(* Logix 5000 project; controller RN21_Architecture 1769-L16ER-BB1B rev 35.11; software revision 35.00; part 5 of 9 *)
(* tags used below, declared in another part *)
   AUDSrc : UDT_Audit;
   RN21_AUD_BAMTrig : DINT[5];
   RN21_AUD_BAT_NTrig : DINT[4];
   RN21_AUD_BAT_PTrig : DINT[4];
   RN21_AUD_NEG_ONS : BOOL[128];
   RN21_AUD_POS_ONS : BOOL[128];
   RN21_AUDBAM_ONS : BOOL[128];
   RN21_Map_BAM : BOOL[128];
   RN21_Map_BAT : BOOL[32];
   RN21_MapBAT_OB : BOOL[128];
(* MainProgram, continued *)

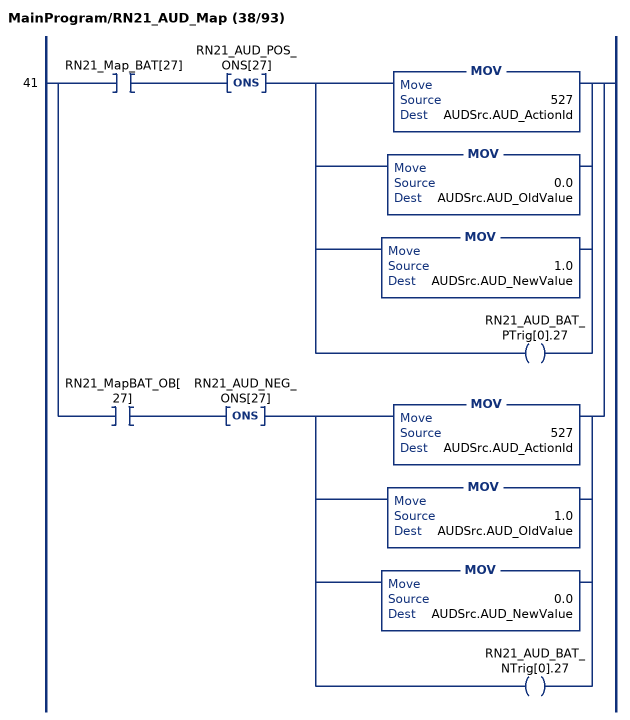
   [picture p120: MainProgram/RN21_AUD_Map rungs 41-41]
   41: [XIC(RN21_Map_BAT[27]) ONS(RN21_AUD_POS_ONS[27]) [MOV(527,AUDSrc.AUD_ActionId) ,MOV(0.0,AUDSrc.AUD_OldValue) ,MOV(1.0,AUDSrc.AUD_NewValue) ,OTE(RN21_AUD_BAT_PTrig[0].27) ] ,XIC(RN21_MapBAT_OB[27]) ONS(RN21_AUD_NEG_ONS[27]) [MOV(527,AUDSrc.AUD_ActionId) ,MOV(1.0,AUDSrc.AUD_OldValue) ,MOV(0.0,AUDSrc.AUD_NewValue) ,OTE(RN21_AUD_BAT_NTrig[0].27) ] ];
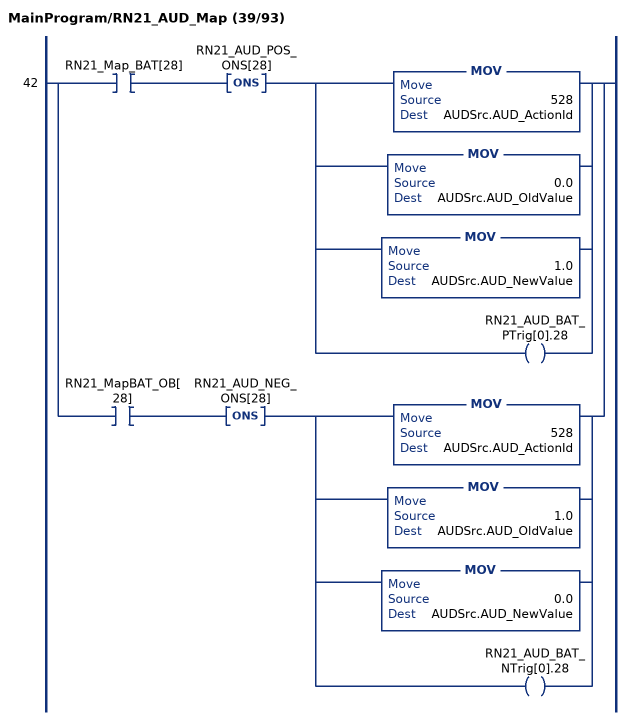
   42: [XIC(RN21_Map_BAT[28]) ONS(RN21_AUD_POS_ONS[28]) [MOV(528,AUDSrc.AUD_ActionId) ,MOV(0.0,AUDSrc.AUD_OldValue) ,MOV(1.0,AUDSrc.AUD_NewValue) ,OTE(RN21_AUD_BAT_PTrig[0].28) ] ,XIC(RN21_MapBAT_OB[28]) ONS(RN21_AUD_NEG_ONS[28]) [MOV(528,AUDSrc.AUD_ActionId) ,MOV(1.0,AUDSrc.AUD_OldValue) ,MOV(0.0,AUDSrc.AUD_NewValue) ,OTE(RN21_AUD_BAT_NTrig[0].28) ] ];
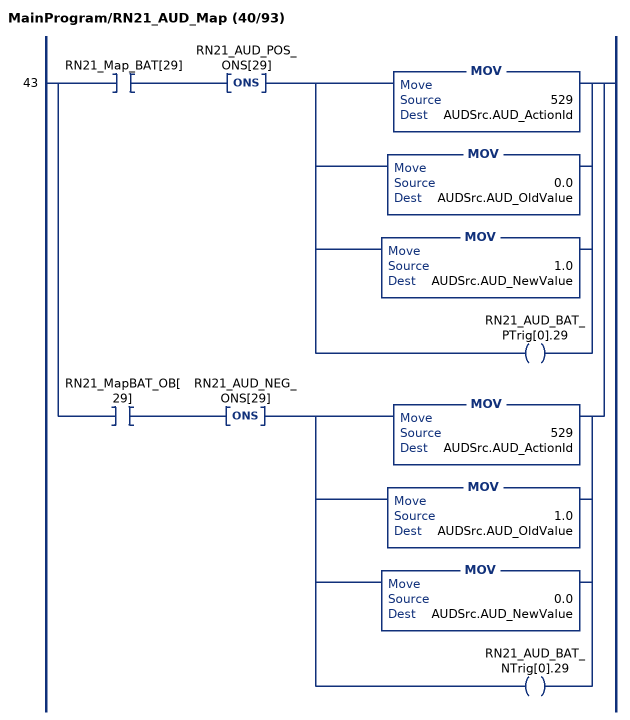
   43: [XIC(RN21_Map_BAT[29]) ONS(RN21_AUD_POS_ONS[29]) [MOV(529,AUDSrc.AUD_ActionId) ,MOV(0.0,AUDSrc.AUD_OldValue) ,MOV(1.0,AUDSrc.AUD_NewValue) ,OTE(RN21_AUD_BAT_PTrig[0].29) ] ,XIC(RN21_MapBAT_OB[29]) ONS(RN21_AUD_NEG_ONS[29]) [MOV(529,AUDSrc.AUD_ActionId) ,MOV(1.0,AUDSrc.AUD_OldValue) ,MOV(0.0,AUDSrc.AUD_NewValue) ,OTE(RN21_AUD_BAT_NTrig[0].29) ] ];
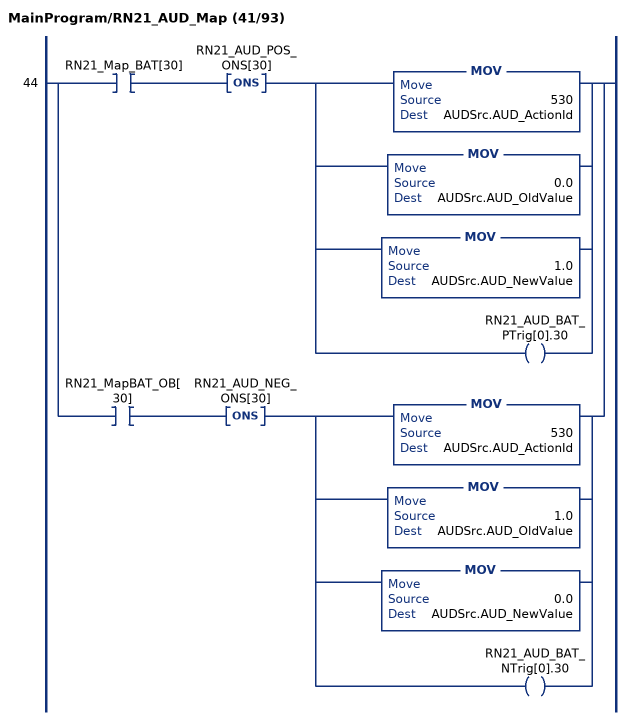
   44: [XIC(RN21_Map_BAT[30]) ONS(RN21_AUD_POS_ONS[30]) [MOV(530,AUDSrc.AUD_ActionId) ,MOV(0.0,AUDSrc.AUD_OldValue) ,MOV(1.0,AUDSrc.AUD_NewValue) ,OTE(RN21_AUD_BAT_PTrig[0].30) ] ,XIC(RN21_MapBAT_OB[30]) ONS(RN21_AUD_NEG_ONS[30]) [MOV(530,AUDSrc.AUD_ActionId) ,MOV(1.0,AUDSrc.AUD_OldValue) ,MOV(0.0,AUDSrc.AUD_NewValue) ,OTE(RN21_AUD_BAT_NTrig[0].30) ] ];
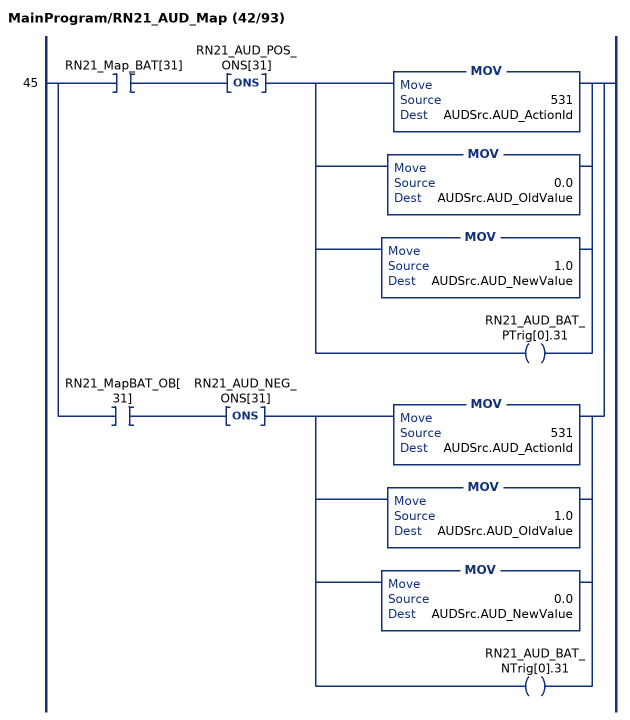
   45: [XIC(RN21_Map_BAT[31]) ONS(RN21_AUD_POS_ONS[31]) [MOV(531,AUDSrc.AUD_ActionId) ,MOV(0.0,AUDSrc.AUD_OldValue) ,MOV(1.0,AUDSrc.AUD_NewValue) ,OTE(RN21_AUD_BAT_PTrig[0].31) ] ,XIC(RN21_MapBAT_OB[31]) ONS(RN21_AUD_NEG_ONS[31]) [MOV(531,AUDSrc.AUD_ActionId) ,MOV(1.0,AUDSrc.AUD_OldValue) ,MOV(0.0,AUDSrc.AUD_NewValue) ,OTE(RN21_AUD_BAT_NTrig[0].31) ] ];
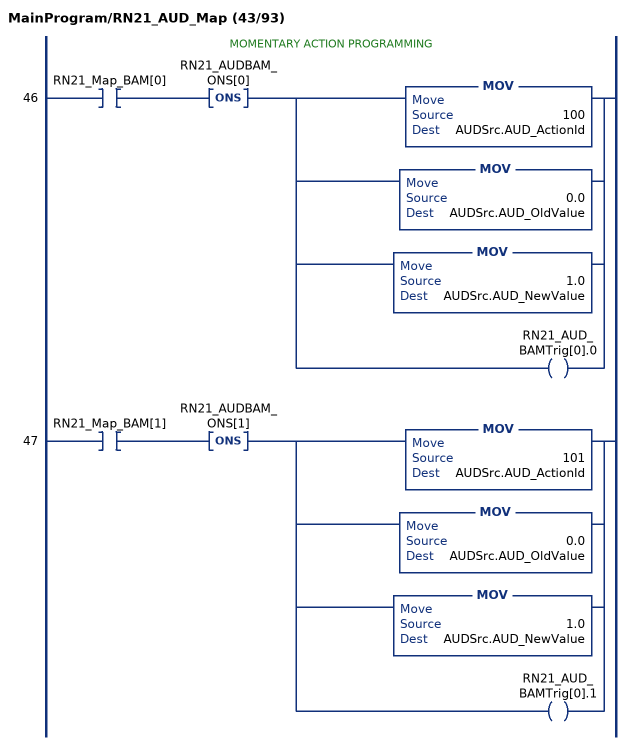
   // MOMENTARY ACTION PROGRAMMING
   46: XIC(RN21_Map_BAM[0])ONS(RN21_AUDBAM_ONS[0])[MOV(100,AUDSrc.AUD_ActionId) ,MOV(0.0,AUDSrc.AUD_OldValue) ,MOV(1.0,AUDSrc.AUD_NewValue) ,OTE(RN21_AUD_BAMTrig[0].0) ];
   47: XIC(RN21_Map_BAM[1])ONS(RN21_AUDBAM_ONS[1])[MOV(101,AUDSrc.AUD_ActionId) ,MOV(0.0,AUDSrc.AUD_OldValue) ,MOV(1.0,AUDSrc.AUD_NewValue) ,OTE(RN21_AUD_BAMTrig[0].1) ];
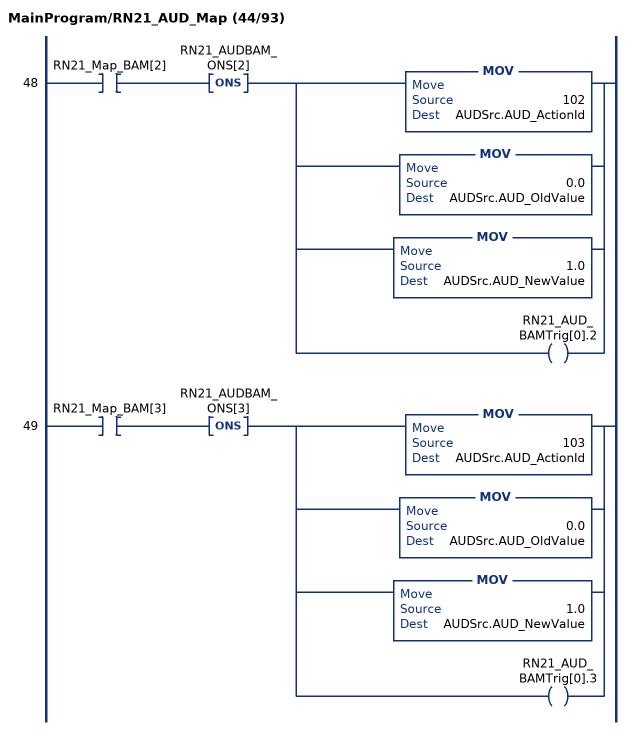
   48: XIC(RN21_Map_BAM[2])ONS(RN21_AUDBAM_ONS[2])[MOV(102,AUDSrc.AUD_ActionId) ,MOV(0.0,AUDSrc.AUD_OldValue) ,MOV(1.0,AUDSrc.AUD_NewValue) ,OTE(RN21_AUD_BAMTrig[0].2) ];
   49: XIC(RN21_Map_BAM[3])ONS(RN21_AUDBAM_ONS[3])[MOV(103,AUDSrc.AUD_ActionId) ,MOV(0.0,AUDSrc.AUD_OldValue) ,MOV(1.0,AUDSrc.AUD_NewValue) ,OTE(RN21_AUD_BAMTrig[0].3) ];
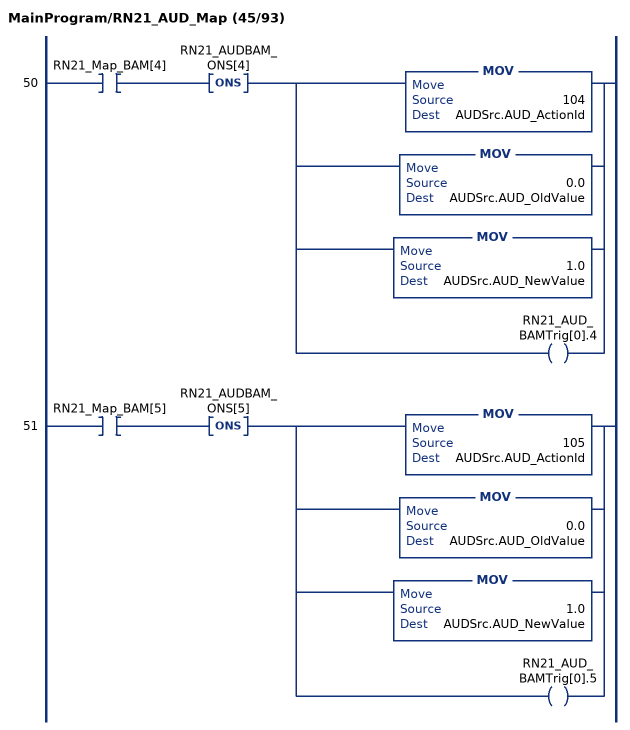
   50: XIC(RN21_Map_BAM[4])ONS(RN21_AUDBAM_ONS[4])[MOV(104,AUDSrc.AUD_ActionId) ,MOV(0.0,AUDSrc.AUD_OldValue) ,MOV(1.0,AUDSrc.AUD_NewValue) ,OTE(RN21_AUD_BAMTrig[0].4) ];
   51: XIC(RN21_Map_BAM[5])ONS(RN21_AUDBAM_ONS[5])[MOV(105,AUDSrc.AUD_ActionId) ,MOV(0.0,AUDSrc.AUD_OldValue) ,MOV(1.0,AUDSrc.AUD_NewValue) ,OTE(RN21_AUD_BAMTrig[0].5) ];
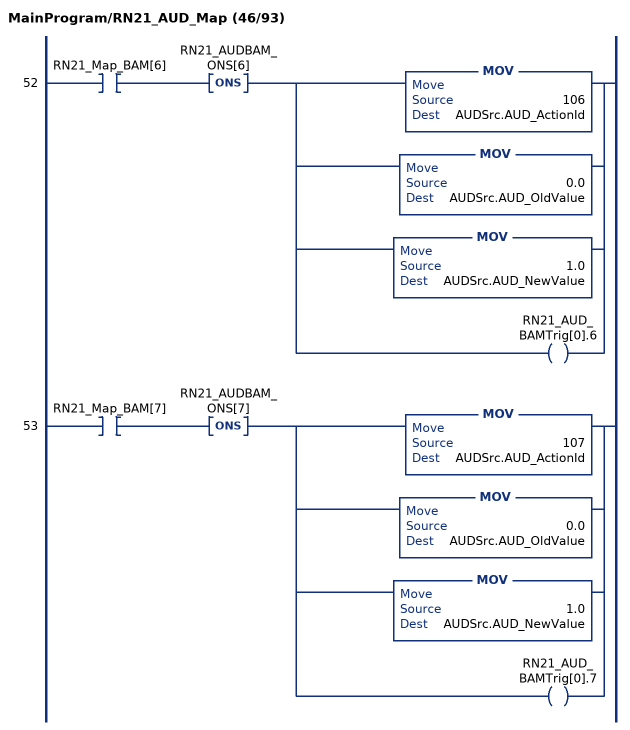
   52: XIC(RN21_Map_BAM[6])ONS(RN21_AUDBAM_ONS[6])[MOV(106,AUDSrc.AUD_ActionId) ,MOV(0.0,AUDSrc.AUD_OldValue) ,MOV(1.0,AUDSrc.AUD_NewValue) ,OTE(RN21_AUD_BAMTrig[0].6) ];
   53: XIC(RN21_Map_BAM[7])ONS(RN21_AUDBAM_ONS[7])[MOV(107,AUDSrc.AUD_ActionId) ,MOV(0.0,AUDSrc.AUD_OldValue) ,MOV(1.0,AUDSrc.AUD_NewValue) ,OTE(RN21_AUD_BAMTrig[0].7) ];
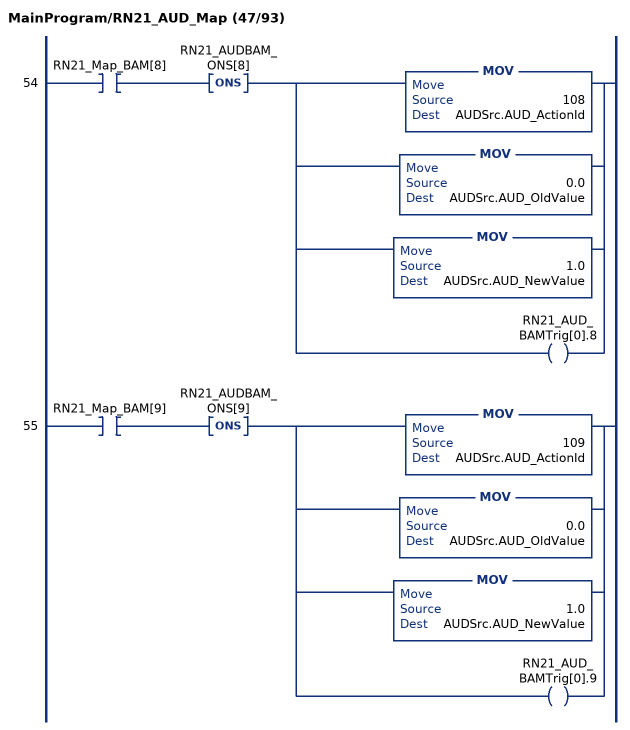
   54: XIC(RN21_Map_BAM[8])ONS(RN21_AUDBAM_ONS[8])[MOV(108,AUDSrc.AUD_ActionId) ,MOV(0.0,AUDSrc.AUD_OldValue) ,MOV(1.0,AUDSrc.AUD_NewValue) ,OTE(RN21_AUD_BAMTrig[0].8) ];
   55: XIC(RN21_Map_BAM[9])ONS(RN21_AUDBAM_ONS[9])[MOV(109,AUDSrc.AUD_ActionId) ,MOV(0.0,AUDSrc.AUD_OldValue) ,MOV(1.0,AUDSrc.AUD_NewValue) ,OTE(RN21_AUD_BAMTrig[0].9) ];
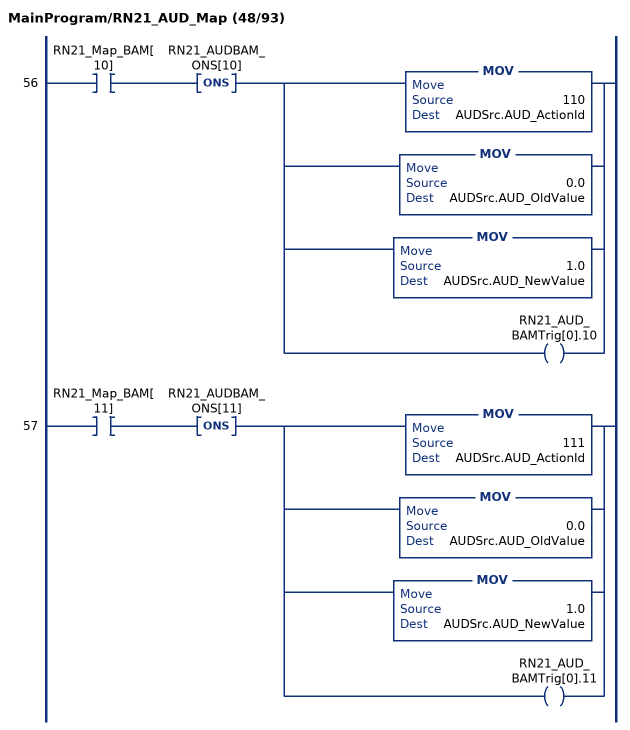
   56: XIC(RN21_Map_BAM[10])ONS(RN21_AUDBAM_ONS[10])[MOV(110,AUDSrc.AUD_ActionId) ,MOV(0.0,AUDSrc.AUD_OldValue) ,MOV(1.0,AUDSrc.AUD_NewValue) ,OTE(RN21_AUD_BAMTrig[0].10) ];
   57: XIC(RN21_Map_BAM[11])ONS(RN21_AUDBAM_ONS[11])[MOV(111,AUDSrc.AUD_ActionId) ,MOV(0.0,AUDSrc.AUD_OldValue) ,MOV(1.0,AUDSrc.AUD_NewValue) ,OTE(RN21_AUD_BAMTrig[0].11) ];
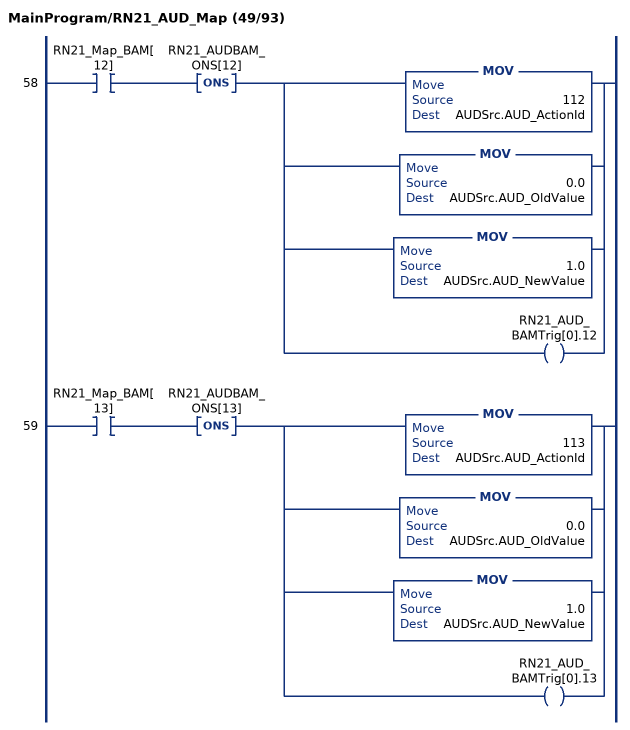
   58: XIC(RN21_Map_BAM[12])ONS(RN21_AUDBAM_ONS[12])[MOV(112,AUDSrc.AUD_ActionId) ,MOV(0.0,AUDSrc.AUD_OldValue) ,MOV(1.0,AUDSrc.AUD_NewValue) ,OTE(RN21_AUD_BAMTrig[0].12) ];
   59: XIC(RN21_Map_BAM[13])ONS(RN21_AUDBAM_ONS[13])[MOV(113,AUDSrc.AUD_ActionId) ,MOV(0.0,AUDSrc.AUD_OldValue) ,MOV(1.0,AUDSrc.AUD_NewValue) ,OTE(RN21_AUD_BAMTrig[0].13) ];
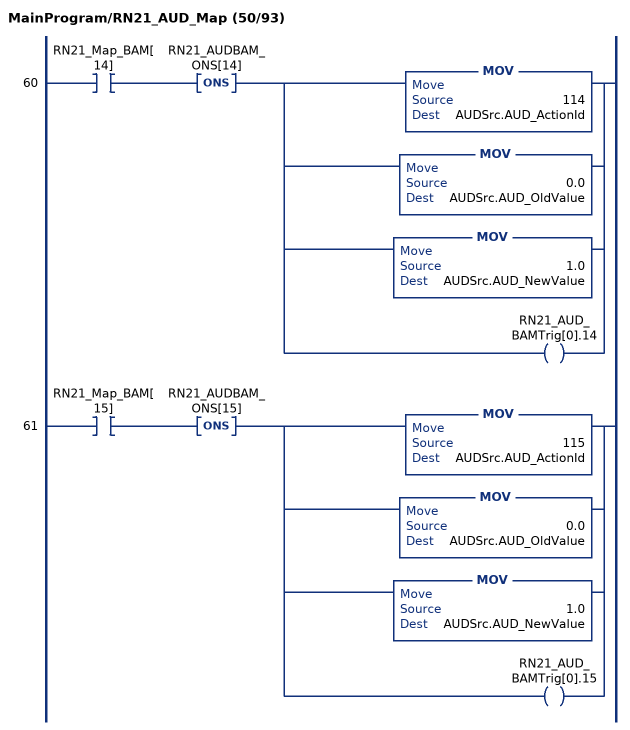
   60: XIC(RN21_Map_BAM[14])ONS(RN21_AUDBAM_ONS[14])[MOV(114,AUDSrc.AUD_ActionId) ,MOV(0.0,AUDSrc.AUD_OldValue) ,MOV(1.0,AUDSrc.AUD_NewValue) ,OTE(RN21_AUD_BAMTrig[0].14) ];
   61: XIC(RN21_Map_BAM[15])ONS(RN21_AUDBAM_ONS[15])[MOV(115,AUDSrc.AUD_ActionId) ,MOV(0.0,AUDSrc.AUD_OldValue) ,MOV(1.0,AUDSrc.AUD_NewValue) ,OTE(RN21_AUD_BAMTrig[0].15) ];
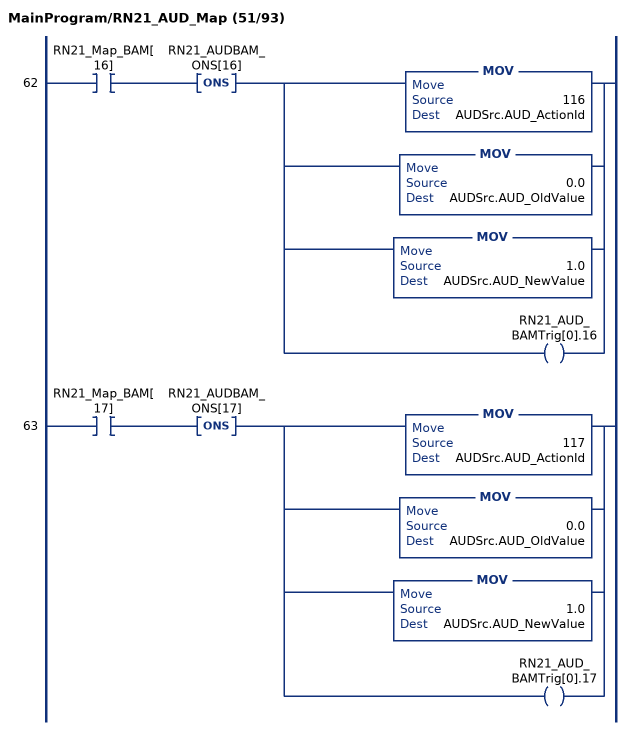
   62: XIC(RN21_Map_BAM[16])ONS(RN21_AUDBAM_ONS[16])[MOV(116,AUDSrc.AUD_ActionId) ,MOV(0.0,AUDSrc.AUD_OldValue) ,MOV(1.0,AUDSrc.AUD_NewValue) ,OTE(RN21_AUD_BAMTrig[0].16) ];
   63: XIC(RN21_Map_BAM[17])ONS(RN21_AUDBAM_ONS[17])[MOV(117,AUDSrc.AUD_ActionId) ,MOV(0.0,AUDSrc.AUD_OldValue) ,MOV(1.0,AUDSrc.AUD_NewValue) ,OTE(RN21_AUD_BAMTrig[0].17) ];
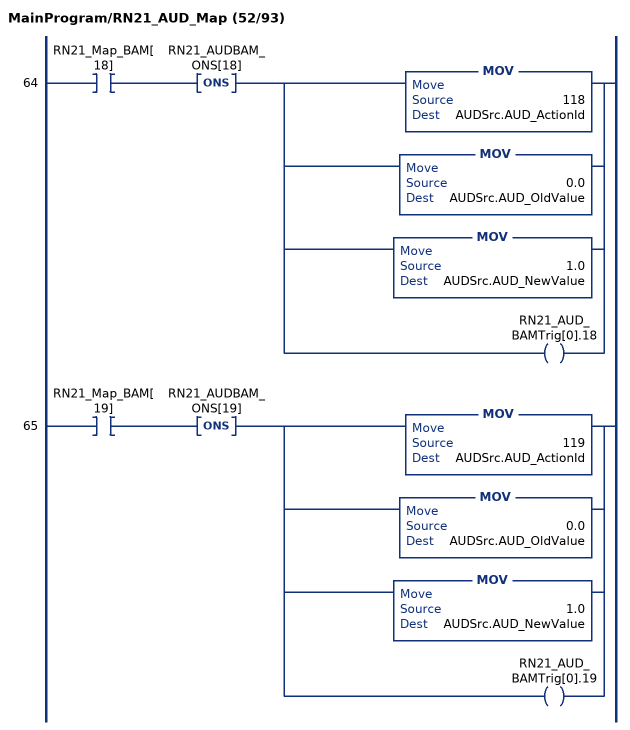
   64: XIC(RN21_Map_BAM[18])ONS(RN21_AUDBAM_ONS[18])[MOV(118,AUDSrc.AUD_ActionId) ,MOV(0.0,AUDSrc.AUD_OldValue) ,MOV(1.0,AUDSrc.AUD_NewValue) ,OTE(RN21_AUD_BAMTrig[0].18) ];
   65: XIC(RN21_Map_BAM[19])ONS(RN21_AUDBAM_ONS[19])[MOV(119,AUDSrc.AUD_ActionId) ,MOV(0.0,AUDSrc.AUD_OldValue) ,MOV(1.0,AUDSrc.AUD_NewValue) ,OTE(RN21_AUD_BAMTrig[0].19) ];
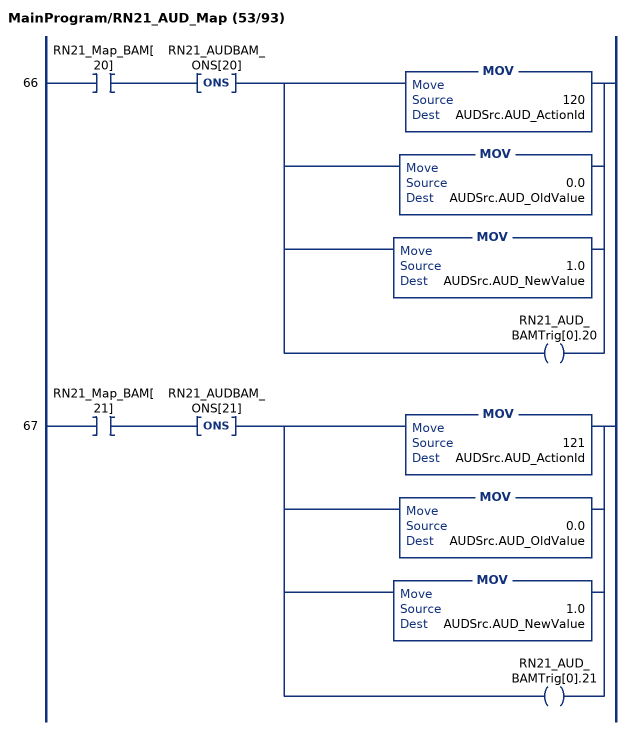
   66: XIC(RN21_Map_BAM[20])ONS(RN21_AUDBAM_ONS[20])[MOV(120,AUDSrc.AUD_ActionId) ,MOV(0.0,AUDSrc.AUD_OldValue) ,MOV(1.0,AUDSrc.AUD_NewValue) ,OTE(RN21_AUD_BAMTrig[0].20) ];
   67: XIC(RN21_Map_BAM[21])ONS(RN21_AUDBAM_ONS[21])[MOV(121,AUDSrc.AUD_ActionId) ,MOV(0.0,AUDSrc.AUD_OldValue) ,MOV(1.0,AUDSrc.AUD_NewValue) ,OTE(RN21_AUD_BAMTrig[0].21) ];
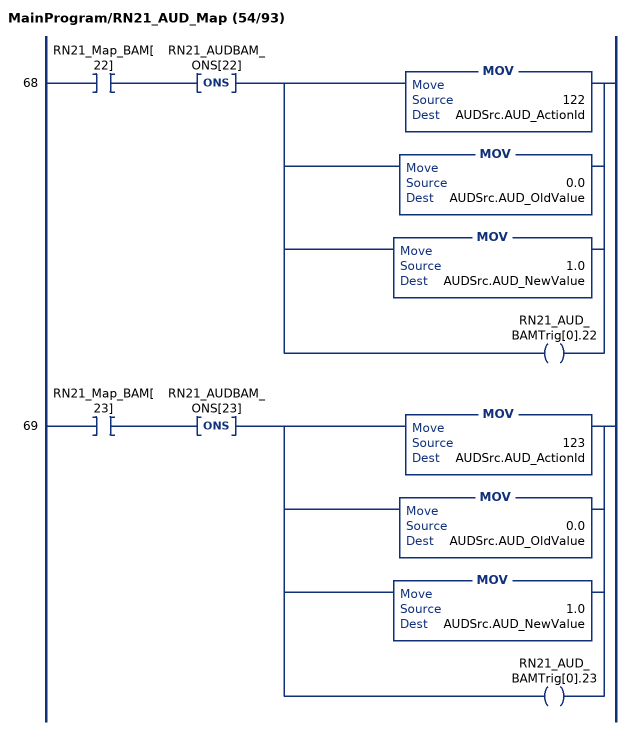
   68: XIC(RN21_Map_BAM[22])ONS(RN21_AUDBAM_ONS[22])[MOV(122,AUDSrc.AUD_ActionId) ,MOV(0.0,AUDSrc.AUD_OldValue) ,MOV(1.0,AUDSrc.AUD_NewValue) ,OTE(RN21_AUD_BAMTrig[0].22) ];
   69: XIC(RN21_Map_BAM[23])ONS(RN21_AUDBAM_ONS[23])[MOV(123,AUDSrc.AUD_ActionId) ,MOV(0.0,AUDSrc.AUD_OldValue) ,MOV(1.0,AUDSrc.AUD_NewValue) ,OTE(RN21_AUD_BAMTrig[0].23) ];
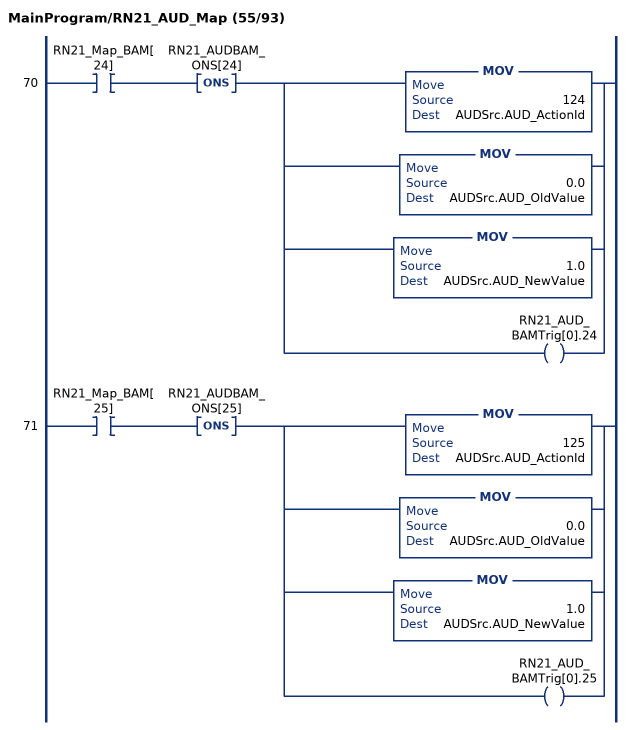
   70: XIC(RN21_Map_BAM[24])ONS(RN21_AUDBAM_ONS[24])[MOV(124,AUDSrc.AUD_ActionId) ,MOV(0.0,AUDSrc.AUD_OldValue) ,MOV(1.0,AUDSrc.AUD_NewValue) ,OTE(RN21_AUD_BAMTrig[0].24) ];
   71: XIC(RN21_Map_BAM[25])ONS(RN21_AUDBAM_ONS[25])[MOV(125,AUDSrc.AUD_ActionId) ,MOV(0.0,AUDSrc.AUD_OldValue) ,MOV(1.0,AUDSrc.AUD_NewValue) ,OTE(RN21_AUD_BAMTrig[0].25) ];
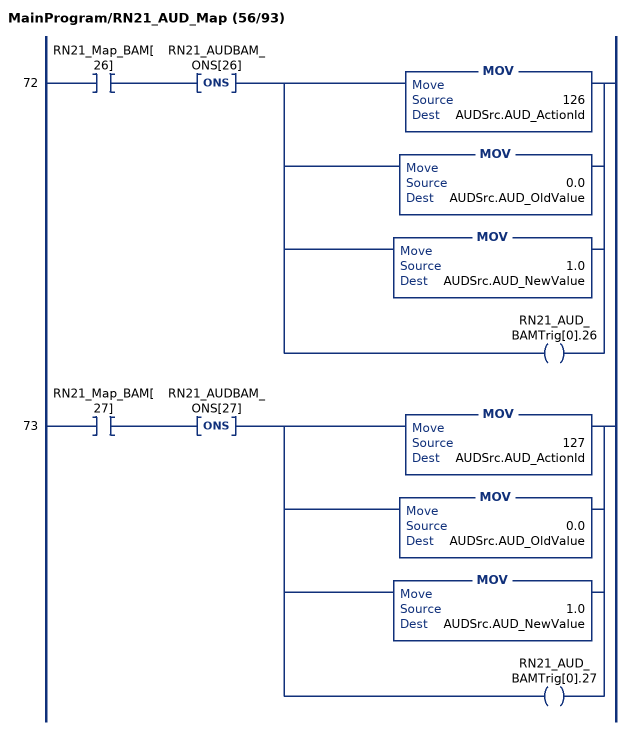
   72: XIC(RN21_Map_BAM[26])ONS(RN21_AUDBAM_ONS[26])[MOV(126,AUDSrc.AUD_ActionId) ,MOV(0.0,AUDSrc.AUD_OldValue) ,MOV(1.0,AUDSrc.AUD_NewValue) ,OTE(RN21_AUD_BAMTrig[0].26) ];
   73: XIC(RN21_Map_BAM[27])ONS(RN21_AUDBAM_ONS[27])[MOV(127,AUDSrc.AUD_ActionId) ,MOV(0.0,AUDSrc.AUD_OldValue) ,MOV(1.0,AUDSrc.AUD_NewValue) ,OTE(RN21_AUD_BAMTrig[0].27) ];
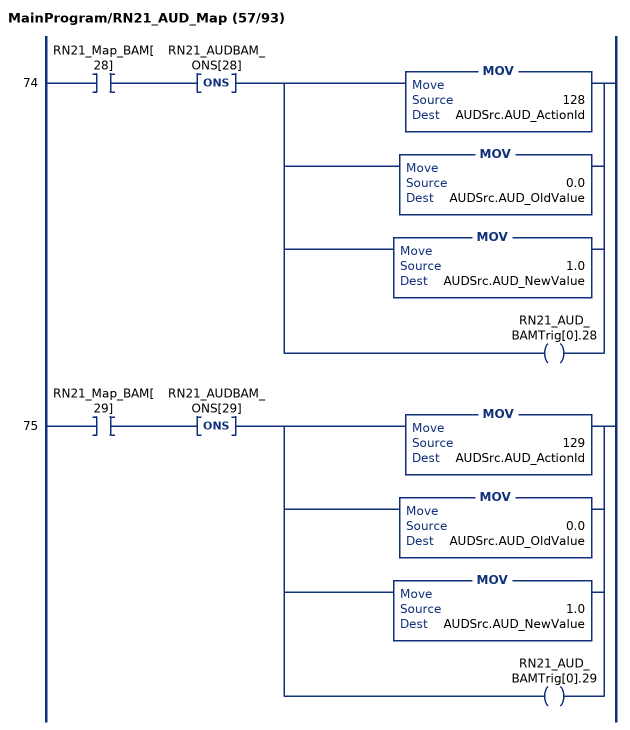
   74: XIC(RN21_Map_BAM[28])ONS(RN21_AUDBAM_ONS[28])[MOV(128,AUDSrc.AUD_ActionId) ,MOV(0.0,AUDSrc.AUD_OldValue) ,MOV(1.0,AUDSrc.AUD_NewValue) ,OTE(RN21_AUD_BAMTrig[0].28) ];
   75: XIC(RN21_Map_BAM[29])ONS(RN21_AUDBAM_ONS[29])[MOV(129,AUDSrc.AUD_ActionId) ,MOV(0.0,AUDSrc.AUD_OldValue) ,MOV(1.0,AUDSrc.AUD_NewValue) ,OTE(RN21_AUD_BAMTrig[0].29) ];
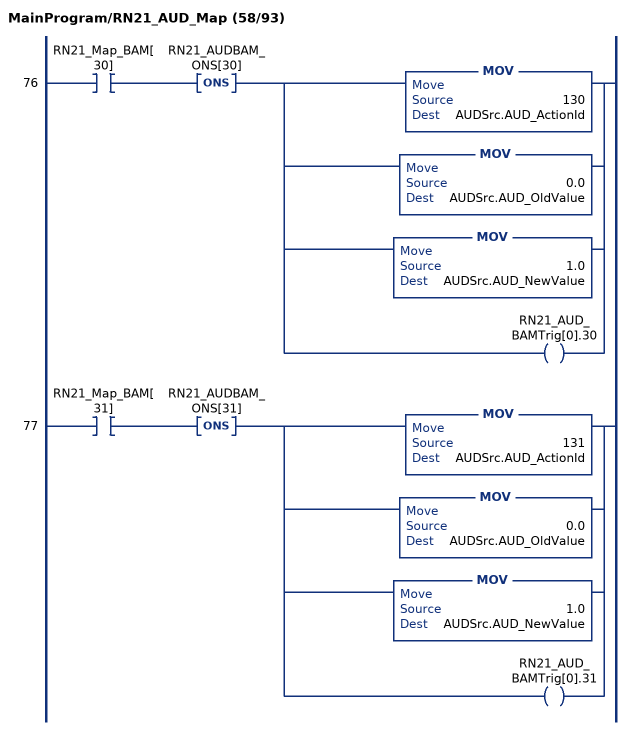
   76: XIC(RN21_Map_BAM[30])ONS(RN21_AUDBAM_ONS[30])[MOV(130,AUDSrc.AUD_ActionId) ,MOV(0.0,AUDSrc.AUD_OldValue) ,MOV(1.0,AUDSrc.AUD_NewValue) ,OTE(RN21_AUD_BAMTrig[0].30) ];
   77: XIC(RN21_Map_BAM[31])ONS(RN21_AUDBAM_ONS[31])[MOV(131,AUDSrc.AUD_ActionId) ,MOV(0.0,AUDSrc.AUD_OldValue) ,MOV(1.0,AUDSrc.AUD_NewValue) ,OTE(RN21_AUD_BAMTrig[0].31) ];
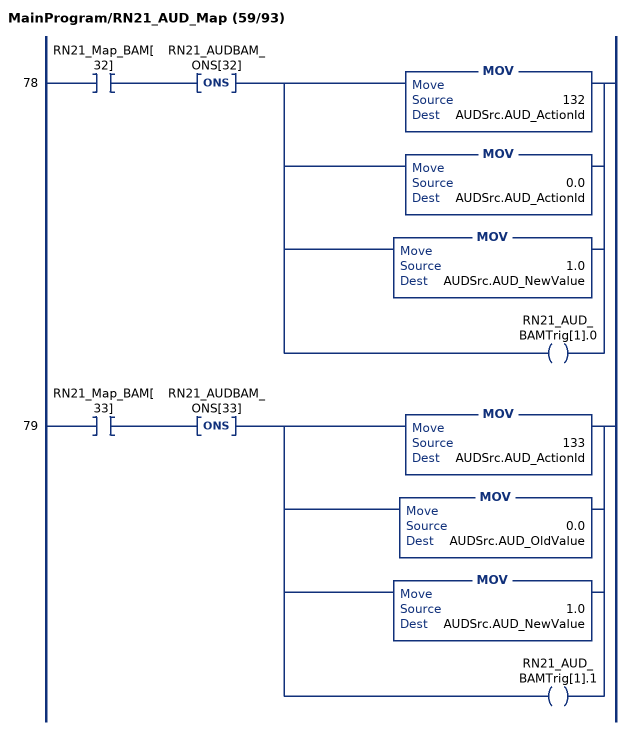
   78: XIC(RN21_Map_BAM[32])ONS(RN21_AUDBAM_ONS[32])[MOV(132,AUDSrc.AUD_ActionId) ,MOV(0.0,AUDSrc.AUD_ActionId) ,MOV(1.0,AUDSrc.AUD_NewValue) ,OTE(RN21_AUD_BAMTrig[1].0) ];
   79: XIC(RN21_Map_BAM[33])ONS(RN21_AUDBAM_ONS[33])[MOV(133,AUDSrc.AUD_ActionId) ,MOV(0.0,AUDSrc.AUD_OldValue) ,MOV(1.0,AUDSrc.AUD_NewValue) ,OTE(RN21_AUD_BAMTrig[1].1) ];
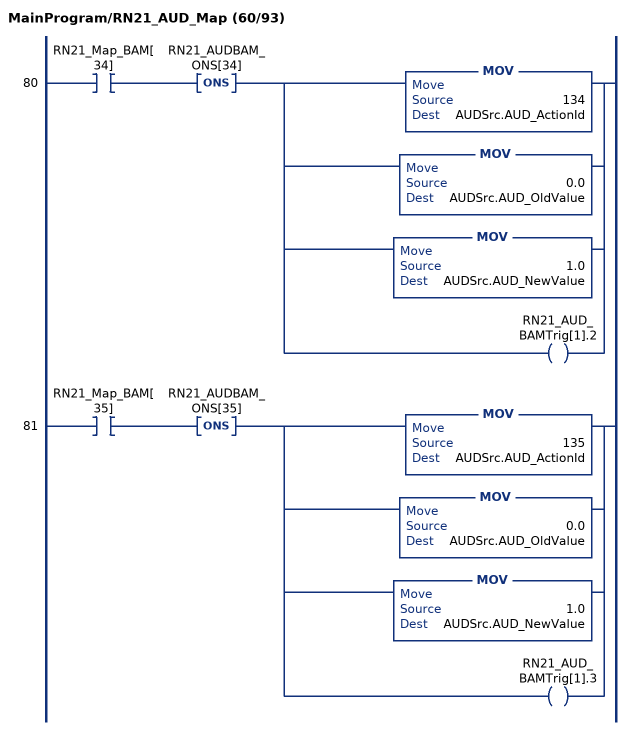
   80: XIC(RN21_Map_BAM[34])ONS(RN21_AUDBAM_ONS[34])[MOV(134,AUDSrc.AUD_ActionId) ,MOV(0.0,AUDSrc.AUD_OldValue) ,MOV(1.0,AUDSrc.AUD_NewValue) ,OTE(RN21_AUD_BAMTrig[1].2) ];
   81: XIC(RN21_Map_BAM[35])ONS(RN21_AUDBAM_ONS[35])[MOV(135,AUDSrc.AUD_ActionId) ,MOV(0.0,AUDSrc.AUD_OldValue) ,MOV(1.0,AUDSrc.AUD_NewValue) ,OTE(RN21_AUD_BAMTrig[1].3) ];
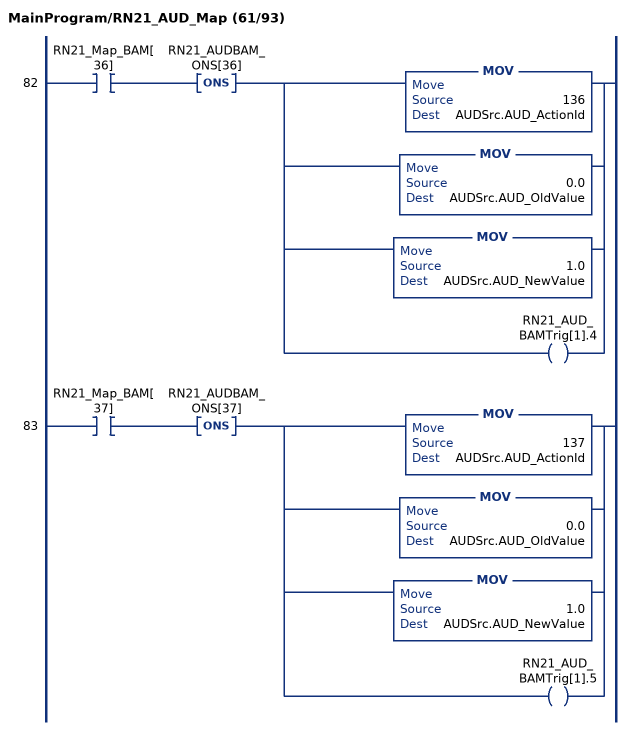
   82: XIC(RN21_Map_BAM[36])ONS(RN21_AUDBAM_ONS[36])[MOV(136,AUDSrc.AUD_ActionId) ,MOV(0.0,AUDSrc.AUD_OldValue) ,MOV(1.0,AUDSrc.AUD_NewValue) ,OTE(RN21_AUD_BAMTrig[1].4) ];
   83: XIC(RN21_Map_BAM[37])ONS(RN21_AUDBAM_ONS[37])[MOV(137,AUDSrc.AUD_ActionId) ,MOV(0.0,AUDSrc.AUD_OldValue) ,MOV(1.0,AUDSrc.AUD_NewValue) ,OTE(RN21_AUD_BAMTrig[1].5) ];
